{attribute 'analysis' := '-33'}
PROGRAM INTERNAL PRG_EnumTests
VAR
{IF defined (UNIT_TEST)}
    fbComputeEnumSizeTests : FB_ComputeEnumSizeTests;
    fbWriteEnumTests       : FB_WriteEnumTests;
    fbReadEnumTests        : FB_ReadEnumTests;
    fbFieldCodecEnumTests  : FB_FieldCodecEnumTests;
{END_IF}
END_VAR

END_PROGRAM

(* stored: Version 1.1.0.1
   POU PRG_EnumTests: Id {ac08c74c-0c17-44f7-bb66-c7967f28da8f}, SpecialFunc None *)
